# EPICS substitutions: ek9000App/Db/EL1008.substitutions
file EL1008.template
{ 	pattern
	{
		TERMINAL,

	}
	{
	}
}
